// TIA Portal V20 export
// export: Created 2025-12-01T14:57:22.6610777Z, ExportSetting None, DisplayName Totally Integrated Automation Portal, DisplayVersion V20 Update 3, DisplayName TIA Portal Openness, DisplayVersion V20 Update 3, DisplayName TIA Portal Version Control Interface, DisplayVersion V20 Update 3, DisplayName STEP 7 Professional, DisplayVersion V20 Update 3, DisplayName STEP 7 Safety, DisplayVersion V20 Update 2, DisplayName WinCC Basic/Comfort/Advanced, DisplayVersion V20 Update 3, DisplayName WinCC Professional, DisplayVersion V20 Update 3, DisplayName WinCC Unified, DisplayVersion V20 Update 3
FUNCTION "FC2_Errores_CCPIF" : Void   // FC2, LAD
{ S7_Optimized_Access := 'FALSE' }
// stored: AutoNumber false, SetENOAutomatically false
BEGIN

REGION Network 1: Activacion de los Emergencias
   // 0 seta 1001
   // 1 seta 1010
   // 2 seta 1020
   // 3 seta 1025
   // 4 seta 1029
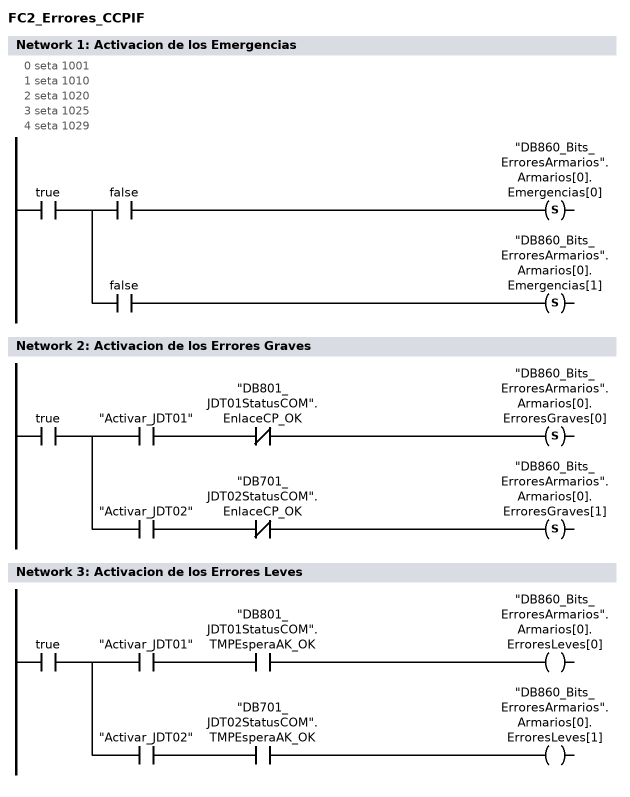
   RUNG wire#powerrail
      Contact( true )
      wire#w1
      Contact( false )
      S_Coil( "DB860_Bits_ErroresArmarios".Armarios[0].Emergencias[0] )
   END_RUNG
   RUNG wire#w1
      Contact( false )
      S_Coil( "DB860_Bits_ErroresArmarios".Armarios[0].Emergencias[1] )
   END_RUNG
   // the same network as SCL:
   IF true AND false THEN
       "DB860_Bits_ErroresArmarios".Armarios[0].Emergencias[0] := TRUE;
       "DB860_Bits_ErroresArmarios".Armarios[0].Emergencias[1] := TRUE;
   END_IF;
END_REGION

REGION Network 2: Activacion de los Errores Graves
   RUNG wire#powerrail
      Contact( true )
      wire#w1
      Contact( "Activar_JDT01" )
      I_Contact( "DB801_JDT01StatusCOM".EnlaceCP_OK )
      S_Coil( "DB860_Bits_ErroresArmarios".Armarios[0].ErroresGraves[0] )
   END_RUNG
   RUNG wire#w1
      Contact( "Activar_JDT02" )
      I_Contact( "DB701_JDT02StatusCOM".EnlaceCP_OK )
      S_Coil( "DB860_Bits_ErroresArmarios".Armarios[0].ErroresGraves[1] )
   END_RUNG
   // the same network as SCL:
   IF true AND "Activar_JDT01" AND NOT "DB801_JDT01StatusCOM".EnlaceCP_OK THEN
       "DB860_Bits_ErroresArmarios".Armarios[0].ErroresGraves[0] := TRUE;
   END_IF;
   IF true AND "Activar_JDT02" AND NOT "DB701_JDT02StatusCOM".EnlaceCP_OK THEN
       "DB860_Bits_ErroresArmarios".Armarios[0].ErroresGraves[1] := TRUE;
   END_IF;
END_REGION

REGION Network 3: Activacion de los Errores Leves
   RUNG wire#powerrail
      Contact( true )
      wire#w1
      Contact( "Activar_JDT01" )
      Contact( "DB801_JDT01StatusCOM".TMPEsperaAK_OK )
      Coil( "DB860_Bits_ErroresArmarios".Armarios[0].ErroresLeves[0] )
   END_RUNG
   RUNG wire#w1
      Contact( "Activar_JDT02" )
      Contact( "DB701_JDT02StatusCOM".TMPEsperaAK_OK )
      Coil( "DB860_Bits_ErroresArmarios".Armarios[0].ErroresLeves[1] )
   END_RUNG
   // the same network as SCL:
   "DB860_Bits_ErroresArmarios".Armarios[0].ErroresLeves[0] := true AND "Activar_JDT01" AND "DB801_JDT01StatusCOM".TMPEsperaAK_OK;
   "DB860_Bits_ErroresArmarios".Armarios[0].ErroresLeves[1] := true AND "Activar_JDT02" AND "DB701_JDT02StatusCOM".TMPEsperaAK_OK;
END_REGION
END_FUNCTION
